ABB RAPID module: RobData.mod

MODULE RobData
    PERS robtarget pPass2:=[[-40.4314,-257.966,143.781],[4.99019E-05,-0.667497,0.744613,6.30517E-05],[-2,-1,-1,0],[9E+09,9E+09,9E+09,9E+09,9E+09,9E+09]];
    PERS robtarget pFcCalib:=[[108.10,-252.03,11.85],[0.000221418,-0.707336,0.706877,0.000273512],[-1,0,0,0],[9E+09,9E+09,9E+09,9E+09,9E+09,9E+09]];
    PERS robtarget phome:=[[-120.88,-372.36,162.78],[0.000481169,-0.706761,0.707452,0.000317998],[-2,-1,-1,0],[9E+09,9E+09,9E+09,9E+09,9E+09,9E+09]];
    PERS robtarget pPlace:=[[-40.42,-221.89,143.77],[1.93875E-05,-0.667481,0.744627,3.37175E-05],[-2,-1,-1,0],[9E+09,9E+09,9E+09,9E+09,9E+09,9E+09]];
	PERS robtarget pPickWait:=[[-119.58,-372.93,143.41],[0.000631318,-0.707272,0.706942,0.000406359],[-2,-1,-1,0],[9E+09,9E+09,9E+09,9E+09,9E+09,9E+09]];
    PERS robtarget pCCD2Cali:=[[227.05,-307.11,144.4],[0.000421342,-0.706769,0.707444,0.000316291],[-1,0,0,0],[9E+09,9E+09,9E+09,9E+09,9E+09,9E+09]];
    PERS robtarget pTCPCalib:=[[28.2702,-315.463,110.616],[0.000286051,-0.259146,-0.965838,-0.000611972],[-1,-1,-3,0],[9E+09,9E+09,9E+09,9E+09,9E+09,9E+09]];
    PERS robtarget pCCD1:=[[27.54,-312.71,110.40],[0.000302404,-0.25914,-0.96584,-0.000644278],[-1,-1,-3,0],[9E+09,9E+09,9E+09,9E+09,9E+09,9E+09]];
	PERS robtarget pPickInkpad:=[[128.85,-272.57,39.17],[0.00042248,-0.706761,0.707452,0.000307461],[-1,0,0,0],[9E+09,9E+09,9E+09,9E+09,9E+09,9E+09]];
    PERS robtarget pPass1:=[[224.96,-305.79,216.82],[0.29997,0.731597,0.298478,-0.534504],[-1,-1,-1,0],[9E+09,9E+09,9E+09,9E+09,9E+09,9E+09]];
    PERS robtarget pPick:=[[-120.88,-372.36,82.78],[0.000481169,-0.706761,0.707452,0.000317998],[-2,-1,-1,0],[9E+09,9E+09,9E+09,9E+09,9E+09,9E+09]];
    PERS robtarget pAssembly:=[[0,0,119],[0,-1,0,0],[-1,0,-1,0],[9E+09,9E+09,9E+09,9E+09,9E+09,9E+09]];
	PERS robtarget pAssem:=[[354.53,109.44,1307.28],[0.522631,-0.494622,0.5135,0.467465],[0,-1,-1,0],[9E+09,9E+09,9E+09,9E+09,9E+09,9E+09]];
    PERS robtarget pInsert:=[[-2.16,-0.09,217.56],[0.0153748,0.716885,-0.0187068,0.69677],[-1,-1,-1,0],[9E+09,9E+09,9E+09,9E+09,9E+09,9E+09]];
    PERS robtarget pAssBase:=[[225.06,-308.31,118.65],[0.0102026,-0.99364,-0.111268,-0.0139692],[-1,0,-1,0],[9E+09,9E+09,9E+09,9E+09,9E+09,9E+09]];
    PERS robtarget pCali2Temp:=[[221.471,-305.943,140.42],[3.87751E-06,0.113366,-0.993553,-6.74824E-05],[-1,0,-1,0],[9E+09,9E+09,9E+09,9E+09,9E+09,9E+09]];
    VAR robtarget pActPos:=[[752.23,113.39,1307.28],[0.522626,-0.494634,0.513503,0.467454],[0,-2,0,0],[9E+09,9E+09,9E+09,9E+09,9E+09,9E+09]];
    PERS tooldata tGripper:=[TRUE,[[0,0,115],[0,0,0,-1]],[1,[0,0,0.001],[1,0,0,0],0,0,0]];
    PERS tooldata tcp1:=[TRUE,[[-134.881,-2.6021,210.993],[0.472574,-0.509839,-0.505206,0.511376]],[0.001,[0,0,0.001],[1,0,0,0],0,0,0]];
    PERS tooldata tcp2:=[TRUE,[[-134.881,-2.6021,210.993],[0.472574,-0.509839,-0.505206,0.511376]],[0.001,[0,0,0.001],[1,0,0,0],0,0,0]];
    PERS tooldata tCurTool:=[TRUE,[[-0.129395,-0.0280151,115],[0.999879,4.09421E-11,-2.3077E-12,0.0155324]],[1,[0,0,0.001],[1,0,0,0],0,0,0]];
    PERS wobjdata AssFrame:=[FALSE,TRUE,"",[[227.265,-307.059,-0.2],[0.504663,0,0,-0.863316]],[[0,0,0],[1,0,0,0]]];
    PERS pose posRel:=[[27.442,-312.621,110.4],[0.000639503,-0.961698,0.274111,0.000312375]];
    !the position of insert action
    PERS robtarget pccd2Calib{9}:=[[[223.05,-311.11,144.4],[0.000421342,-0.706769,0.707444,0.000316291],[-1,0,0,0],[9E+09,9E+09,9E+09,9E+09,9E+09,9E+09]],[[223.05,-307.11,144.4],[0.000421342,-0.706769,0.707444,0.000316291],[-1,0,0,0],[9E+09,9E+09,9E+09,9E+09,9E+09,9E+09]],[[223.05,-303.11,144.4],[0.000421342,-0.706769,0.707444,0.000316291],[-1,0,0,0],[9E+09,9E+09,9E+09,9E+09,9E+09,9E+09]],[[227.05,-311.11,144.4],[0.000421342,-0.706769,0.707444,0.000316291],[-1,0,0,0],[9E+09,9E+09,9E+09,9E+09,9E+09,9E+09]],[[227.05,-307.11,144.4],[0.000421342,-0.706769,0.707444,0.000316291],[-1,0,0,0],[9E+09,9E+09,9E+09,9E+09,9E+09,9E+09]],[[227.05,-303.11,144.4],[0.000421342,-0.706769,0.707444,0.000316291],[-1,0,0,0],[9E+09,9E+09,9E+09,9E+09,9E+09,9E+09]],[[231.05,-311.11,144.4],[0.000421342,-0.706769,0.707444,0.000316291],[-1,0,0,0],[9E+09,9E+09,9E+09,9E+09,9E+09,9E+09]],[[231.05,-307.11,144.4],[0.000421342,-0.706769,0.707444,0.000316291],[-1,0,0,0],[9E+09,9E+09,9E+09,9E+09,9E+09,9E+09]],[[231.05,-303.11,144.4],[0.000421342,-0.706769,0.707444,0.000316291],[-1,0,0,0],[9E+09,9E+09,9E+09,9E+09,9E+09,9E+09]]];
    CONST robtarget p10:=[[418.58,0.00,334.20],[0.69977,-5.36606E-06,0.714368,-1.01452E-05],[-1,-1,-1,1],[9E+09,9E+09,9E+09,9E+09,9E+09,9E+09]];
	CONST robtarget p20:=[[-0.78,-0.98,134.97],[0.045115,-0.778366,0.0549846,-0.623769],[-1,-1,-1,0],[9E+09,9E+09,9E+09,9E+09,9E+09,9E+09]];
	CONST robtarget p30:=[[3.25,-1.23,131.34],[0.052365,-0.893272,0.0373206,-0.444893],[-1,-1,-1,0],[9E+09,9E+09,9E+09,9E+09,9E+09,9E+09]];
	CONST robtarget p40:=[[7.31,-1.27,127.32],[0.0574813,-0.964587,0.0229531,-0.256401],[-1,-1,-1,0],[9E+09,9E+09,9E+09,9E+09,9E+09,9E+09]];
	CONST robtarget p50:=[[6.55,1.54,127.33],[0.0250852,-0.966495,-0.128089,-0.221022],[-1,-1,-1,0],[9E+09,9E+09,9E+09,9E+09,9E+09,9E+09]];
	CONST robtarget p60:=[[4.98,0.64,125.42],[0.0167574,-0.97874,-0.129439,-0.158219],[-1,-1,-1,0],[9E+09,9E+09,9E+09,9E+09,9E+09,9E+09]];
	CONST robtarget p70:=[[3.86,4.82,125.54],[0.0207843,0.921285,0.354866,0.157707],[-1,-1,-2,0],[9E+09,9E+09,9E+09,9E+09,9E+09,9E+09]];
	CONST robtarget p80:=[[3.90,4.13,124.94],[0.0541693,-0.873114,-0.472372,-0.107716],[-1,-1,-2,0],[9E+09,9E+09,9E+09,9E+09,9E+09,9E+09]];
	CONST robtarget p90:=[[-0.27,1.56,123.30],[0.00352402,-0.711908,-0.701467,-0.0334439],[-1,-1,-3,0],[9E+09,9E+09,9E+09,9E+09,9E+09,9E+09]];
	CONST robtarget p100:=[[4.30,1.38,122.36],[0.0190123,-0.977767,-0.196515,-0.07065],[-1,-1,-2,0],[9E+09,9E+09,9E+09,9E+09,9E+09,9E+09]];
	CONST robtarget p110:=[[4.73,3.47,122.36],[0.00254348,0.877137,0.474635,0.0731187],[-1,-1,-2,0],[9E+09,9E+09,9E+09,9E+09,9E+09,9E+09]];
	CONST robtarget p120:=[[2.48,3.22,122.00],[0.00800762,0.838824,0.543446,0.0312499],[-1,-1,-2,0],[9E+09,9E+09,9E+09,9E+09,9E+09,9E+09]];
	CONST robtarget p130:=[[0.78,0.99,121.75],[0.0133946,0.729882,0.682811,0.0293496],[-1,-1,-3,0],[9E+09,9E+09,9E+09,9E+09,9E+09,9E+09]];
	CONST robtarget p140:=[[395.07,52.94,69.21],[0.146773,-0.40343,-0.902897,-0.0218841],[0,0,0,0],[9E+09,9E+09,9E+09,9E+09,9E+09,9E+09]];
	CONST robtarget p150:=[[0.73,0.19,121.74],[0.00247764,0.730292,0.683065,0.00947357],[-1,-1,-3,0],[9E+09,9E+09,9E+09,9E+09,9E+09,9E+09]];
	CONST robtarget p160:=[[0.62,3.16,122.50],[0.0216987,-0.999509,-0.0111852,0.0196521],[-1,-1,-1,0],[9E+09,9E+09,9E+09,9E+09,9E+09,9E+09]];
	CONST robtarget p170:=[[0.15,1.60,122.60],[0.022889,-0.999681,-0.0106178,-0.00147162],[-1,0,-1,0],[9E+09,9E+09,9E+09,9E+09,9E+09,9E+09]];
	CONST robtarget p180:=[[0.33,0.75,122.56],[0.0405975,-0.99906,-0.000325195,-0.0151796],[-1,0,-1,0],[9E+09,9E+09,9E+09,9E+09,9E+09,9E+09]];
	CONST robtarget p190:=[[-5.04,9.32,128.15],[0.502915,0.733369,-0.411451,-0.199886],[-1,-1,0,0],[9E+09,9E+09,9E+09,9E+09,9E+09,9E+09]];
	CONST robtarget p200:=[[-7.89,9.59,127.41],[0.377726,0.806199,-0.437126,-0.127621],[-1,-1,0,0],[9E+09,9E+09,9E+09,9E+09,9E+09,9E+09]];
	CONST robtarget p210:=[[309.31,-185.13,57.93],[3.23688E-05,-0.711176,0.703014,2.50774E-05],[-1,0,-2,0],[9E+09,9E+09,9E+09,9E+09,9E+09,9E+09]];
	CONST robtarget p220:=[[309.31,-185.13,60.13],[3.17998E-05,-0.71117,0.70302,2.71847E-05],[-1,0,-2,0],[9E+09,9E+09,9E+09,9E+09,9E+09,9E+09]];
    CONST robtarget p230:=[[291.17,-178.69,59.38],[0.121864,0.177542,0.974817,-0.0579603],[-1,-1,0,0],[9E+09,9E+09,9E+09,9E+09,9E+09,9E+09]];
	CONST robtarget p240:=[[291.17,-178.69,59.38],[0.0237281,0.143256,0.987655,-0.0587628],[-1,-1,0,0],[9E+09,9E+09,9E+09,9E+09,9E+09,9E+09]];
	CONST robtarget p250:=[[294.50,-178.67,59.37],[0.0180936,0.0502125,0.996728,-0.0607034],[-1,-1,-1,0],[9E+09,9E+09,9E+09,9E+09,9E+09,9E+09]];
	CONST robtarget p260:=[[296.33,-183.75,59.37],[0.00909617,-0.0948952,0.99347,-0.0626853],[-1,-1,-1,0],[9E+09,9E+09,9E+09,9E+09,9E+09,9E+09]];
	CONST robtarget p270:=[[299.47,-185.58,56.25],[0.0201912,0.533122,-0.843665,0.060031],[-1,-1,-1,0],[9E+09,9E+09,9E+09,9E+09,9E+09,9E+09]];
	CONST robtarget p280:=[[309.31,-185.13,57.93],[3.23688E-05,-0.711176,0.703014,2.50774E-05],[-1,0,-2,0],[9E+09,9E+09,9E+09,9E+09,9E+09,9E+09]];
	CONST robtarget p290:=[[309.31,-185.13,60.13],[3.17998E-05,-0.71117,0.70302,2.71847E-05],[-1,0,-2,0],[9E+09,9E+09,9E+09,9E+09,9E+09,9E+09]];
    VAR jointtarget J_Temp:=[[0,0,0,0,0,0],[0,0,0,0,0,0]];
    PERS string sCCD;
    PERS string Revision:="Rev 3.3.2";
    PERS string sFirstStr;
    PERS string sSecondStr;
    PERS num Zangle:=-96.2604;
    PERS num Yangle:=-0.00782723;
    PERS num Xangle:=179.998;
    VAR string CCD1X{9}:=["","","","","","","","",""];
    VAR string CCD1Y{9}:=["","","","","","","","",""];
    VAR string CCD2X{9}:=["","","","","","","","",""];
    VAR string CCD2Y{9}:=["","","","","","","","",""];
    PERS NUM ARRAY{9}:=[3,6,9,8,5,2,1,4,7];
    VAR string sCCD1;
    VAR string sCCD3;
    PERS num nanglex:=0;
    PERS num nangley:=0;
    !CCD 1 data for pick the Buttun
    PERS num X1:=27.442;
    PERS num Y1:=-312.621;
    PERS num nAngle1:=-32.218;
    !CCD2 data for gasket
    PERS num X2:=227.265;
    PERS num Y2:=-307.059;
    PERS num nAngle2:=-29.382;
    !CCD3 data for cable;
    PERS num X3:=-1.1567;
    PERS num Y3:=0;
    PERS num nAngle3:=0;
    PERS num X4:=35.818;
    PERS num Y4:=-312.359;
    PERS num nAngle4:=1.27;
    !the data from computer to modify the robot position

    !CCD3 data for cable;
    PERS num noffsX:=-0.27;
    PERS num noffsY:=-0.67;
    PERS num noffsAngle:=0.4;
    PERS num nAssX:=0.3;
    PERS num nAssY:=0;
    PERS num nAssz:=-0.2;
    PERS num XC:=9;
    PERS num YC:=20;
    PERS num nCCD:=0;
    PERS num nccd3offs:=0;
    PERS num nccd3offsx:=0;
    PERS num nTempX:=-5;
    PERS num nTempY:=0;
    PERS num nTempZ:=0;
    PERS num nTAnglez:=0;
    PERS num nTAngley:=0;
    PERS num nTAnglex:=0;
    PERS num nPositionNo:=0;
    PERS num nHtemp:=0;
    !the insert speed of the robot
    PERS speeddata vAssembly:=[200,25,5000,1000];
    PERS num baseX2:=0;
    PERS num baseY2:=0;
    PERS bool bFull:=TRUE;
    PERS bool bWork:=FALSE;
    PERS bool bCalibration:=FALSE;
    PERS bool bInitall:=FALSE;
    PERS bool bEmptyDone:=FALSE;
    PERS bool SockGet:=FALSE;
    VAR intnum iSocketError:=0;
    VAR intnum iCalibration:=0;
    VAR intnum iInitall:=0;
    VAR intnum iEmptydone:=0;
    VAR intnum iProcessFinish:=0;
    !CCD3 data for
    PERS num CCD1_X:=425.2;
    PERS num CCD1_Y:=-118.686;
    PERS num AngZ:=0;
    !Gasket wobj Z value

    VAR socketdev temp_socket;
    PERS tooldata tGrip:=[TRUE,[[0,0,108],[1,0,0,0]],[2,[0,1,0],[1,0,0,0],0,0,0]];
    PERS tooldata tTCP:=[TRUE,[[0,0,120],[1,0,0,0]],[2,[0,1,0],[1,0,0,0],0,0,0]];
    PERS num n:=2;
    PERS num b:=3;
    PERS num nStrLength:=10;
    PERS num nfind:=6;
    PERS num nArray{20}:=[6,20,29,37,45,54,20,23,26,29,5,8,11,14,17,20,23,26,0,0];
    var num nArray1{9}:=[13,20,29,37,45,54,59,66,73];
    var num nArray2{3}:=[11,18,0];
    PERS pose nPoseAss:=[[0,-0.3,-0.2],[1,0,0,0]];
    PERS pos nPOSCCD1{9}:=[[23.5381,-314.928,110.622],[23.541,-312.732,110.618],[23.5407,-310.532,110.618],[27.5395,-314.924,110.621],[27.5425,-312.733,110.619],[27.5408,-310.533,110.62],[31.5414,-314.929,110.623],[31.5425,-312.733,110.619],[31.5417,-310.532,110.618]];
    PERS pos nPOSCCD2{9}:=[[225.056,-305.11,144.394],[227.053,-305.109,144.392],[229.055,-305.114,144.395],[229.054,-307.111,144.392],[227.055,-307.114,144.394],[225.053,-307.111,144.393],[225.054,-309.113,144.392],[227.055,-309.111,144.394],[229.054,-309.111,144.396]];
    PERS String SocketStr:="startpress";
    PERS String SendStr:="";
    PERS String sFrame:="world";
    CONST robtarget p300:=[[35.94,-312.18,78.08],[0.0367958,-0.00985026,-0.999273,0.00150693],[-1,-1,-1,0],[9E+09,9E+09,9E+09,9E+09,9E+09,9E+09]];
    PERS robtarget pCCD1Cali:=[[27.54,-312.71,110.40],[0.000302404,-0.25914,-0.96584,-0.000644278],[-1,-1,-3,0],[9E+09,9E+09,9E+09,9E+09,9E+09,9E+09]];
    PERS robtarget pccd2Calib_T{9}:=[[[225.05,-309.11,144.4],[0.000421342,-0.706769,0.707444,0.000316291],[-1,0,0,0],[9E+09,9E+09,9E+09,9E+09,9E+09,9E+09]],[[225.05,-307.11,144.4],[0.000421342,-0.706769,0.707444,0.000316291],[-1,0,0,0],[9E+09,9E+09,9E+09,9E+09,9E+09,9E+09]],[[225.05,-305.11,144.4],[0.000421342,-0.706769,0.707444,0.000316291],[-1,0,0,0],[9E+09,9E+09,9E+09,9E+09,9E+09,9E+09]],[[227.05,-309.11,144.4],[0.000421342,-0.706769,0.707444,0.000316291],[-1,0,0,0],[9E+09,9E+09,9E+09,9E+09,9E+09,9E+09]],[[227.05,-307.11,144.4],[0.000421342,-0.706769,0.707444,0.000316291],[-1,0,0,0],[9E+09,9E+09,9E+09,9E+09,9E+09,9E+09]],[[227.05,-305.11,144.4],[0.000421342,-0.706769,0.707444,0.000316291],[-1,0,0,0],[9E+09,9E+09,9E+09,9E+09,9E+09,9E+09]],[[229.05,-309.11,144.4],[0.000421342,-0.706769,0.707444,0.000316291],[-1,0,0,0],[9E+09,9E+09,9E+09,9E+09,9E+09,9E+09]],[[229.05,-307.11,144.4],[0.000421342,-0.706769,0.707444,0.000316291],[-1,0,0,0],[9E+09,9E+09,9E+09,9E+09,9E+09,9E+09]],[[229.05,-305.11,144.4],[0.000421342,-0.706769,0.707444,0.000316291],[-1,0,0,0],[9E+09,9E+09,9E+09,9E+09,9E+09,9E+09]]];
    VAR intnum intDoor:=0;
    PERS wobjdata AssFrame1:=[FALSE,TRUE,"",[[227.265,-307.059,-0.2],[0.967308,0,0,-0.253606]],[[0,0,0],[1,0,0,0]]];
ENDMODULE
